TYPE ST_pValveDeadBand :
STRUCT
	fPosMax	: LREAL := 29460; // Positive min value [19660..29490]
	fPosMin	: LREAL := 19660; // Positive max value [19660..29490]
	fNegMin : LREAL := 19660; // Negative max value [9830..19660]
	fNegMax	: LREAL := 9830; // Negative min value [9830..19660]
END_STRUCT
END_TYPE

(* stored: Version 1.1.0.1, ProductVersion 3.1.4024.12
   DUT ST_pValveDeadBand: Id {0492f17c-a257-420a-a357-c8c70bfcd085} *)
